Staubli VAL3: GetCutLength.pgx

public program GetCutLength(point& x_pCut[], point& x_pMC[], bool& x_bMC[], num& x_nLength, bool& x_bRes)
  local num l_nNum
  local trsf l_trBuff[3]
  local trsf l_trTe
  local num l_nArc
begin
  //获得切割的真正长度是多少



  x_bRes=false
  x_nLength=0
  if size(x_pCut)!=size(x_pMC) or size(x_pCut)!=size(x_bMC)
    return
  endIf

  //如果只有一个点，则退出
   if size(x_bMC)==1
    x_bRes=true
    return
  endIf


  //多于一个点进行计算
  for l_nNum=1 to size(x_bMC)-1


    if !x_bMC[l_nNum]
      x_nLength=distance(x_pCut[l_nNum-1].trsf,x_pCut[l_nNum].trsf)+x_nLength

    else
      l_trBuff[0]=x_pCut[l_nNum-1].trsf
      l_trBuff[1]=x_pMC[l_nNum].trsf
      l_trBuff[2]=x_pCut[l_nNum].trsf
      //获取圆弧长度
      call GetArcLength(l_trBuff,l_nArc,x_bRes)
      if !x_bRes
        return
      endIf
      x_nLength=x_nLength+l_nArc

    endIf


  endFor

  x_bRes=true

end
